KUKA KRL data list: masref_main.dat

&ACCESS RVO1
&REL 3
&COMMENT Mastering Reference Main Task
&PARAM DISKPATH = KRC:\R1\Program\System
&PARAM EDITMASK = *
DEFDAT  MasRef_Main
;FOLD EXTERNAL DECLARATIONS;%{PE}%MKUKATPBASIS,%CEXT,%VCOMMON,%P
;FOLD GRIPPERTECH EXT
  EXT  H50 (INT:IN, INT:IN ,INT:IN ,GRP_TYP:IN)
;ENDFOLD (GRIPPERTECH EXT)
;FOLD SPOTTECH EXT
  EXT  USERSPOT (S_COMMAND  :IN, SPOT_TYPE:IN)
;ENDFOLD (SPOTTECH EXT)
;FOLD BASISTECH EXT;%{PE}%MKUKATPBASIS,%CEXT,%VEXT,%P
  EXT  BAS (BAS_COMMAND  :IN,REAL  :IN )
;ENDFOLD (BASISTECH EXT)
;FOLD USER EXT;%{E}%MKUKATPUSER,%CEXT,%VEXT,%P
;ENDFOLD (USER EXT)
;ENDFOLD (EXTERNAL DECLERATIONS)
INT nLapsedTime
INT nLapsedTimeout=30
INT PerformMasterReference=0; index for $flag to trigger mastering reference
ENDDAT
